TYPE ST_HexMove_Output :
STRUCT
	Disp_P: matrix_18_real_T;
END_STRUCT
END_TYPE

(* stored: Version 1.1.0.1, ProductVersion 3.1.4020.12
   DUT ST_HexMove_Output: Id {84ec5c55-0870-49a7-9ca1-e69e771f196a} *)
